FUNCTION TryConvert_UINT_TO_STRING : BOOL
VAR_INPUT
	in : UINT;
	out : REFERENCE TO STRING;
END_VAR

out := UINT_TO_STRING(in);
TryConvert_UINT_TO_STRING := TRUE;

END_FUNCTION

(* stored: Version 1.1.0.1, ProductVersion 3.1.4024.12
   POU TryConvert_UINT_TO_STRING: Id {ad775777-bf08-4501-86b5-d581acb59a4e}, SpecialFunc None *)
